FUNCTION_BLOCK fb_operationEjector
VAR_INPUT
END_VAR
VAR_OUTPUT
END_VAR
VAR
	SFCInit : bool;
	flgInitDone: BOOL;
	trn_vacuumOnDone: BOOL;
	trn_vacuumOffDone: BOOL;
	trn_breakOnDone: BOOL;
	trn_breakOffDone: BOOL;
	var_process: INT;
END_VAR

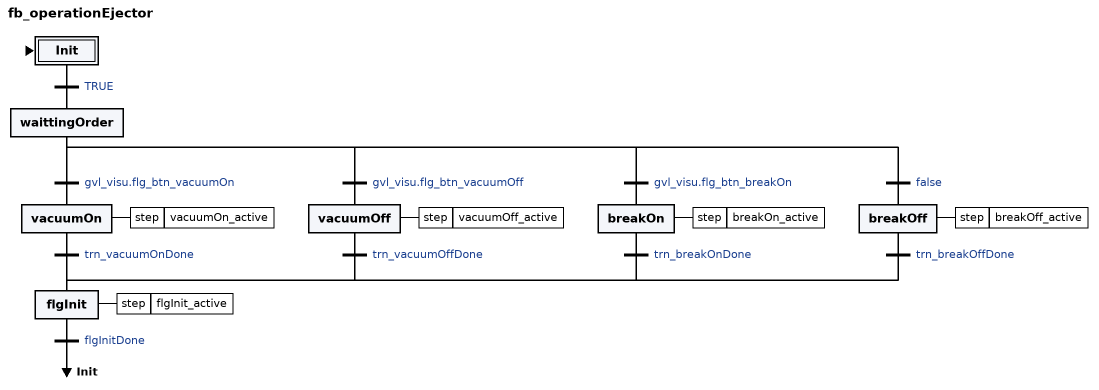
INITIAL_STEP Init:
END_STEP
TRANSITION FROM Init TO waittingOrder
    := TRUE;
END_TRANSITION
STEP waittingOrder:
END_STEP
TRANSITION FROM waittingOrder TO vacuumOn
    := gvl_visu.flg_btn_vacuumOn;
END_TRANSITION
STEP vacuumOn:
    vacuumOn_active(N);  // step action
END_STEP
TRANSITION FROM vacuumOn TO flgInit
    := trn_vacuumOnDone;
END_TRANSITION
TRANSITION FROM waittingOrder TO vacuumOff
    := gvl_visu.flg_btn_vacuumOff;
END_TRANSITION
STEP vacuumOff:
    vacuumOff_active(N);  // step action
END_STEP
TRANSITION FROM vacuumOff TO flgInit
    := trn_vacuumOffDone;
END_TRANSITION
TRANSITION FROM waittingOrder TO breakOn
    := gvl_visu.flg_btn_breakOn;
END_TRANSITION
STEP breakOn:
    breakOn_active(N);  // step action
END_STEP
TRANSITION FROM breakOn TO flgInit
    := trn_breakOnDone;
END_TRANSITION
TRANSITION FROM waittingOrder TO breakOff
    := false;
END_TRANSITION
STEP breakOff:
    breakOff_active(N);  // step action
END_STEP
TRANSITION FROM breakOff TO flgInit
    := trn_breakOffDone;
END_TRANSITION
STEP flgInit:
    flgInit_active(N);  // step action
END_STEP
TRANSITION FROM flgInit TO Init
    := flgInitDone;
END_TRANSITION

ACTION breakOff_active:
IF breakOff._x AND breakOff.x = FALSE THEN
	trn_breakOffDone := FALSE;
	gvl_solv.fbi_ejector.in_flg_run := FALSE;
	gvl_solv.fbi_ejector.in_var_vacMode := eP_ejevacMode.breakOff;
	var_process := 0;
ELSIF breakOff._x AND breakOff.x THEN
	CASE var_process OF
		0:
			gvl_solv.fbi_ejector.in_flg_run := TRUE;
			var_process := 1;
		1:
			IF gvl_solv.fbi_ejector.out_flg_Done THEN
				gvl_solv.fbi_ejector.in_flg_run := FALSE;
				trn_breakOffDone := TRUE;
			END_IF
	END_CASE
END_IF
END_ACTION

ACTION breakOn_active:
IF breakOn._x AND breakOn.x = FALSE THEN
	trn_breakOnDone := FALSE;
	gvl_solv.fbi_ejector.in_flg_run := FALSE;
	gvl_solv.fbi_ejector.in_var_vacMode := eP_ejevacMode.break;
	var_process := 0;
ELSIF breakOn._x AND breakOn._x THEN
	CASE var_process OF
		0:
			gvl_solv.fbi_ejector.in_flg_run := TRUE;
			var_process := 1;
		1:
			IF gvl_solv.fbi_ejector.out_flg_Done THEN
				gvl_solv.fbi_ejector.in_flg_run := FALSE;
				trn_breakOnDone := TRUE;
			END_IF
	END_CASE
END_IF
END_ACTION

ACTION flgInit_active:
IF flgInit._x AND flgInit.x = FALSE THEN
	flgInitDone := FALSE;
	gvl_visu.flg_btn_vacuumOn := FALSE;
	gvl_visu.flg_btn_vacuumOff := FALSE;
	gvl_visu.flg_btn_breakOn := FALSE;
	
ELSIF flgInit._x AND flgInit.x THEN
	flgInitDone := TRUE;
END_IF
END_ACTION

PROPERTY p_Init : bool
GET
p_init := THIS^.SFCInit;
END_GET
SET
THIS^.SFCInit := p_Init;
END_SET
END_PROPERTY

ACTION vacuumOff_active:
IF vacuumOff._x AND vacuumOff.x = FALSE THEN
	trn_vacuumOffDone := FALSE;
	gvl_solv.fbi_ejector.in_flg_run := FALSE;
	gvl_solv.fbi_ejector.in_var_vacMode := eP_ejevacMode.vacOff;
	var_process := 0;
ELSIF vacuumOff._x AND vacuumOff.x THEN
	CASE var_process OF
		0:
			gvl_solv.fbi_ejector.in_flg_run := TRUE;
			var_process :=1;
		1:
			IF gvl_solv.fbi_ejector.out_flg_Done THEN
				gvl_solv.fbi_ejector.in_flg_run := FALSE;
				trn_vacuumOffDone := TRUE;
			END_IF
	END_CASE
END_IF
END_ACTION

ACTION vacuumOn_active:
IF vacuumOn._x AND vacuumOn.x = FALSE THEN
	trn_vacuumOnDone := FALSE;
	gvl_solv.fbi_ejector.in_flg_run := FALSE;
	gvl_solv.fbi_ejector.in_var_vacMode := eP_ejevacMode.halt;
	var_process := 0;
ELSIF vacuumOn._x AND vacuumOn.x THEN
	CASE var_process OF
		0:
			gvl_solv.fbi_ejector.in_flg_run := TRUE;
			var_process := 1;
		1:
			IF gvl_solv.fbi_ejector.out_flg_Done THEN
				gvl_solv.fbi_ejector.in_flg_run := FALSE;
				trn_vacuumOnDone := TRUE;
			END_IF
	END_CASE
END_IF
END_ACTION

END_FUNCTION_BLOCK

(* stored: Version 1.1.0.1, ProductVersion 3.1.4024.11
   POU fb_operationEjector: Id {49e7ccd6-a1b0-41f7-81b4-734588808feb}, SpecialFunc None
   Action breakOff_active: Id {fdbcb606-122f-4b26-a31a-025c2a0506de}
   Action breakOn_active: Id {60138123-8aca-4e4b-8de3-e91e6c5b944e}
   Action flgInit_active: Id {fd2f796e-5866-455d-bd89-7c6cbdec739a}
   Property p_Init: Id {02501365-d0fb-4441-94e7-003607c03182}
   Get Get: Id {6b51d58b-616f-4ce2-a12f-93b2b4c84f2b}
   Set Set: Id {661bd528-831a-458f-8567-9c2084aa69b8}
   Action vacuumOff_active: Id {0268d05d-f94c-4825-8e74-532b8d094ca0}
   Action vacuumOn_active: Id {491e8fea-30bd-4e52-a6ab-eba0f304b82b} *)
